% RSLogix 500 project I2P-JOB-24 DUNCAN_SUTTON_BAK080.RSS, saved by version 10.00.00.00 %
PROJECT "ML01A"    % processor: Bul.1763 MicroLogix 1100 Series B %

PROGRAM FILES
  LAD 2   3 rungs

DATA FILES
  O0 OUTPUT  4 elements
  I1 INPUT  6 elements
  S2 STATUS  66 elements
  B3 BINARY  2 elements
  T4 TIMER  3 elements
  C5 COUNTER  4 elements
  R6 CONTROL  1 elements
  N7 INTEGER  1 elements
  F8 FLOAT  1 elements

LADDER 2
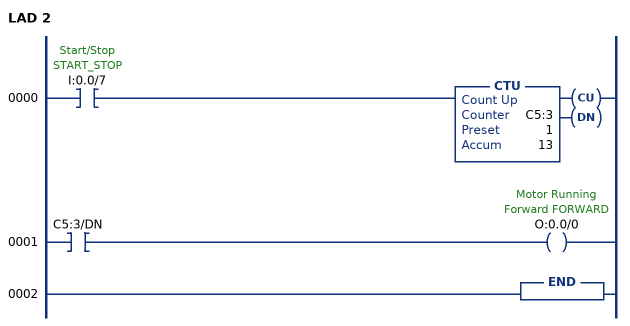
% Rung: 0 %
SOR XIC I:0.0/7 CTU C5:3 1 13 EOR
%   I:0.0/7  START_STOP  "Start/Stop" %
% Rung: 1 %
SOR XIC C5:3/DN OTE O:0.0/0 EOR
%   O:0.0/0  FORWARD  "Motor Running Forward" %
% Rung: 2 %
SOR END EOR

OTHER DOCUMENTED ADDRESSES
  B3:0/0  B_START  "Start"
  B3:0/1  B_FWD  "FWD Memory"
  B3:0/2  B_REV  "Reverse Memory"
  B3:0/3  LAST_FWD  "Memory Direction Foward"
  B3:0/4  LAST_REV  "Memory Direction Reverse"
  B3:0/8  START  "Memory Start"
  B3:0/9  STOP  "Memory Stop"
  C5:0  MTRF_OV  "Motor Forwards OverClock"
  C5:1  MTRR_OV  "Motor Reverse OverClock"
  C5:2/DN  START_UP
  I:0.0/0  ESTOP  "Emergency Stop"
  I:0.0/1  MSF_STAT  "Motor Starter Status (Forwards)"
  I:0.0/2  MSR_STAT  "Motor Starter Status (Reverse)"
  I:0.0/3  FWD  "Direction Motor Forwards"
  I:0.0/4  REV  "Direction Motor Reverse"
  I:0.0/5  MODE  "Mode: A=Run B=Jog"
  I:0.0/6  S  "Stop Motor"
  I:0.0/8  RESET  "Reset Start Counters"
  I:0.0/9  MS_OL  "Motor Overload Contacts"
  I:0.1  MS
  O:0.0/1  OVERLOAD  "Motor Overload"
  O:0.0/2  STOPPED  "Motor Stopped"
  O:0.0/3  REVERSE  "Motor Running Reverse"
  O:0.0/4  MS_F  "Motor Contactor Forwards"
  O:0.0/5  MS_R  "Motor Contactor Reverse"
  T4:0  MTR_CD  "Motor Cool-Down Time"
  T4:0.ACC  MTR_CD_S  "Motor Cool-Down Time Signal"
  T4:0.ACC/0  T4
  T4:0.ACC/6  DIR_CHN  "Direction Change"
  T4:0.PRE  OVERCLOCK  "Collective Motor OverClock"
  T4:0/DN  CMT_DN  "Collective Motor Run Time Done"
  T4:0/TT  MTR_CD_TT  "Motor Cool-Down Wait Action"
  T4:1  MCT_F  "Motor Collective Run Time Forwards"
  T4:1/DN  MCTF_DN  "Motor Collectve Forwards Done"
  T4:2  MCT_R  "Motor Collective Run Time Reverse"
  T4:2/DN  MCTR_DN  "Motor Collective Reverse Done"

DATA TABLE (non-zero values as saved)
DATA T4
% .PRE .ACC %
% T4:0 % 800 0
% T4:1 % 32767 0
% T4:2 % 32767 0
DATA C5
% .PRE .ACC %
% C5:2 % 1 0
% C5:3 % 1 13
